FUNCTION_BLOCK E_PERMIT (* Permissive propagation of an event (synthetic test fixture) *)
  PACKAGE IEC61499.Standard;
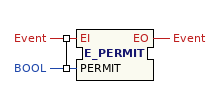
  EVENT_INPUT
    EI WITH PERMIT;
  END_EVENT
  EVENT_OUTPUT
    EO;
  END_EVENT
  VAR_INPUT
    PERMIT : BOOL;
  END_VAR
END_FUNCTION_BLOCK
